KUKA KRL program: dai_sen_calibrate_01.src, dai_sen_calibrate_01.dat

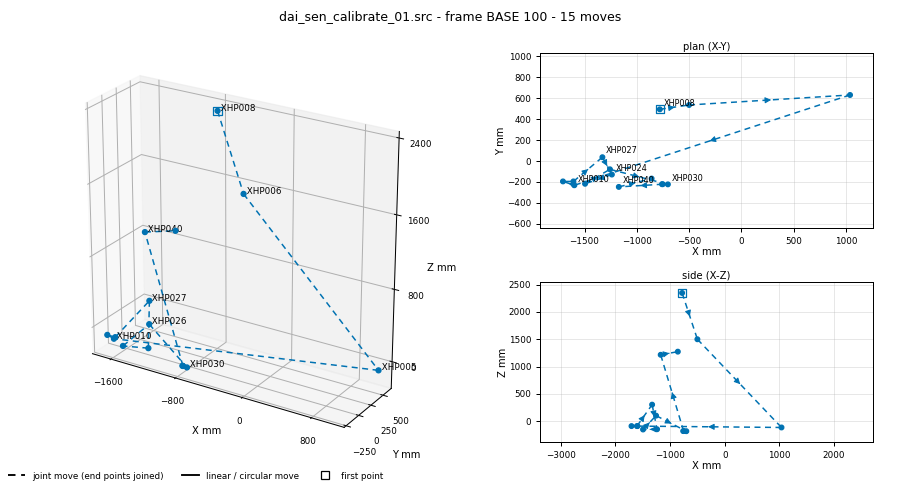
[picture p0: tool path of dai_sen_calibrate_01.src in frame BASE 100, 15 of 17 moves have a stored position in this frame; points joined in program order, loops and branches not executed]
--- dai_sen_calibrate_01.src ---
&ACCESS RVP
&REL 74
&COMMENT Sensopart Kalibrierung
&PARAM TEMPLATE = C:\KRC\roboter\template\vg_appl
&PARAM DISKPATH = KRC:\R1\H_Prog
DEF dai_sen_calibrate_01( )
;FOLD INI;%{PE}
  ;FOLD BASISTECH INI
    GLOBAL INTERRUPT DECL 3 WHEN $STOPMESS==TRUE DO IR_STOPM ( )
    INTERRUPT ON 3
    BAS (#INITMOV,0 )
  ;ENDFOLD (BASISTECH INI)
  ;FOLD USER INI
    ;Make your modifications here
  ;ENDFOLD (USER INI)
;ENDFOLD (INI)
;FOLD ; Anlagenbezeichn: HC51_C    Stations-Nr: 080RB_100;%{PE}
;FOLD Parameters ;%{h}
;Params IlfProvider=kukaroboter.basistech.inlineforms.comments.comment; Kuka.Content=Anlagenbezeichn: HC51_C    Stations-Nr: 080RB_100
;ENDFOLD
;ENDFOLD
;FOLD ; Stand / Version: V1.0;%{PE}
;FOLD Parameters ;%{h}
;Params IlfProvider=kukaroboter.basistech.inlineforms.comments.comment; Kuka.Content=Stand / Version: V1.0
;ENDFOLD
;ENDFOLD
;FOLD ; Name Bearbeiter: EBZ-AE;%{PE}
;FOLD Parameters ;%{h}
;Params IlfProvider=kukaroboter.basistech.inlineforms.comments.comment; Kuka.Content=Name Bearbeiter: EBZ-AE
;ENDFOLD
;ENDFOLD
;FOLD ; Translator Version:29.01.2024 - Version 15.08;%{PE}
;FOLD Parameters ;%{h}
;Params IlfProvider=kukaroboter.basistech.inlineforms.comments.comment; Kuka.Content=Translator Version:29.01.2024 - Version 15.08
;ENDFOLD
;ENDFOLD

;check program once again after mounting calibration plate
WAIT FOR FALSE ;STATUS
;PROGRAM CHECKED BY: SZALA

REPEAT

;FOLD MSG_T1
MSG_SHOW("DAI_H_Prog",#quit,999,"dai_rob_ok_0")
;ENDFOLD

; ***************************************
; A C H T U N G !!! Nur in $T1 abfahren
; ***************************************
UNTIL $T1 == TRUE

REPEAT

;FOLD MSG_T1
MSG_SHOW("DAI_H_Prog",#quit,999,"dai_rob_ok_0")
;ENDFOLD

; ***************************************
; A C H T U N G !!! Nur in $T1 abfahren
; ***************************************
UNTIL $T1 == TRUE

;FOLD PTP HOME Vel=100 % DEFAULT;%{PE}
;FOLD Parameters ;%{h}
;Params IlfProvider=kukaroboter.basistech.inlineforms.movement.old; Kuka.IsGlobalPoint=False; Kuka.PointName=HOME; Kuka.BlendingEnabled=False; Kuka.MoveDataPtpName=DEFAULT; Kuka.VelocityPtp=100; Kuka.CurrentCDSetIndex=0; Kuka.MovementParameterFieldEnabled=True; IlfCommand=PTP
;ENDFOLD
$BWDSTART = FALSE
PDAT_ACT = PDEFAULT
FDAT_ACT = FHOME
BAS(#PTP_PARAMS, 100.0)
SET_CD_PARAMS (0)
PTP XHOME
;ENDFOLD

;Dynamische Pruefung Teil vorhanden
;FOLD PartPresent.CheckOff #1:5279, #2:5280, #3:1025, #4:1025, #5:1025, #6:1025, Bounce Time:100, Constant: Yes;%{PE}%
CheckPartPresent(5279,5280,1025,1025,1025,1025,100, True,FALSE)
;ENDFOLD

;Greifer-Ventile betatigen/pruefen
;FOLD DAI_GripValveCheck.Valve2 State:Fixierstift Ausfahren Gs, 080GRH101-QM1;%{PE}%
CheckValveState(2,1)
;ENDFOLD
;FOLD DAI_GripValveCheck.Valve3 State:Spanner Oeffnen Gs, 080GRH101-QM2;%{PE}%
CheckValveState(3,1)
;ENDFOLD
;FOLD DAI_GripValveCheck.Valve4 State:Sauger Abblasen Gs, 080GRH101-QM3;%{PE}%
CheckValveState(4,1)
;ENDFOLD
;FOLD DAI_GripValveCheck.Valve5 State:Sauger Abblasen Gs, 080GRH101-QM4;%{PE}%
CheckValveState(5,1)
;ENDFOLD

;FOLD PTP HP008 CONT Vel=100 % PDAT16 Tool[110]:MSK_01_XYa_Sensopart Base[100]:SENSOPART_CALIBRATEPLATE ;%{PE}
;FOLD Parameters ;%{h}
;Params IlfProvider=kukaroboter.basistech.inlineforms.movement.old; Kuka.IsGlobalPoint=False; Kuka.PointName=HP008; Kuka.BlendingEnabled=True; Kuka.MoveDataPtpName=PDAT16; Kuka.VelocityPtp=100; Kuka.CurrentCDSetIndex=0; Kuka.MovementParameterFieldEnabled=True; IlfCommand=PTP
;ENDFOLD
$BWDSTART = FALSE
PDAT_ACT = PPDAT16
FDAT_ACT = FHP008
BAS(#PTP_PARAMS, 100.0)
SET_CD_PARAMS (0)
PTP XHP008 C_Dis
;ENDFOLD
;FOLD PTP HP006 CONT Vel=100 % PDAT4 Tool[110]:MSK_01_XYa_Sensopart Base[100]:SENSOPART_CALIBRATEPLATE ;%{PE}
;FOLD Parameters ;%{h}
;Params IlfProvider=kukaroboter.basistech.inlineforms.movement.old; Kuka.IsGlobalPoint=False; Kuka.PointName=HP006; Kuka.BlendingEnabled=True; Kuka.MoveDataPtpName=PDAT4; Kuka.VelocityPtp=100; Kuka.CurrentCDSetIndex=0; Kuka.MovementParameterFieldEnabled=True; IlfCommand=PTP
;ENDFOLD
$BWDSTART = FALSE
PDAT_ACT = PPDAT4
FDAT_ACT = FHP006
BAS(#PTP_PARAMS, 100.0)
SET_CD_PARAMS (0)
PTP XHP006 C_Dis
;ENDFOLD
;FOLD PTP HP005 CONT Vel=100 % PDAT2 Tool[110]:MSK_01_XYa_Sensopart Base[100]:SENSOPART_CALIBRATEPLATE ;%{PE}
;FOLD Parameters ;%{h}
;Params IlfProvider=kukaroboter.basistech.inlineforms.movement.old; Kuka.IsGlobalPoint=False; Kuka.PointName=HP005; Kuka.BlendingEnabled=True; Kuka.MoveDataPtpName=PDAT2; Kuka.VelocityPtp=100; Kuka.CurrentCDSetIndex=0; Kuka.MovementParameterFieldEnabled=True; IlfCommand=PTP
;ENDFOLD
$BWDSTART = FALSE
PDAT_ACT = PPDAT2
FDAT_ACT = FHP005
BAS(#PTP_PARAMS, 100.0)
SET_CD_PARAMS (0)
PTP XHP005 C_Dis
;ENDFOLD

;FOLD PTP HP010 Vel=100 % PDAT3 Tool[110]:MSK_01_XYa_Sensopart Base[100]:SENSOPART_CALIBRATEPLATE ;%{PE}
;FOLD Parameters ;%{h}
;Params IlfProvider=kukaroboter.basistech.inlineforms.movement.old; Kuka.IsGlobalPoint=False; Kuka.PointName=HP010; Kuka.BlendingEnabled=False; Kuka.MoveDataPtpName=PDAT3; Kuka.VelocityPtp=100; Kuka.CurrentCDSetIndex=0; Kuka.MovementParameterFieldEnabled=True; IlfCommand=PTP
;ENDFOLD
$BWDSTART = FALSE
PDAT_ACT = PPDAT3
FDAT_ACT = FHP010
BAS(#PTP_PARAMS, 100.0)
SET_CD_PARAMS (0)
PTP XHP010
;ENDFOLD

;Kalibrationposition
;Fokus-Abstand Kamera zur Kalibrierplatte xx0mm
;FOLD LIN SEN520W080_005 Vel=0.2 m/s CPDAT4 Tool[110]:MSK_01_XYa_Sensopart Base[100]:SENSOPART_CALIBRATEPLATE ;%{PE}
;FOLD Parameters ;%{h}
;Params IlfProvider=kukaroboter.basistech.inlineforms.movement.old; Kuka.IsGlobalPoint=False; Kuka.PointName=SEN520W080_005; Kuka.BlendingEnabled=False; Kuka.MoveDataName=CPDAT4; Kuka.VelocityPath=0.2; Kuka.CurrentCDSetIndex=0; Kuka.MovementParameterFieldEnabled=True; IlfCommand=LIN
;ENDFOLD
$BWDSTART = FALSE
LDAT_ACT = LCPDAT4
FDAT_ACT = FSEN520W080_005
BAS(#CP_PARAMS, 0.2)
SET_CD_PARAMS (0)
LIN XSEN520W080_005
;ENDFOLD

;;FOLD DAI_SEN.CHANGEJOB Cam: 1, Job nbr.: 1 ;%{PE}
; SEN_Cam=1
; SEN_JobResponse=1
; DAI_SEN_CMD ( #ChangeJob )
;;ENDFOLD
;;FOLD DAI_SEN.CALIBRATION Cam: 1, Calibration Base/Tool: 30, Waiting Time: 1 s ;%{PE}
; SEN_CalibMode=2
; SEN_JobResponse=1
; SEN_TimeOut=1
; SEN_CalibBase=30
; SEN_Cam=1
; SEN_CopyMode=1
; DAI_SEN_CMD ( #CALIBRATION )
;;ENDFOLD

;FOLD LIN HP015 Vel=0.2 m/s CPDAT5 Tool[110]:MSK_01_XYa_Sensopart Base[100]:SENSOPART_CALIBRATEPLATE ;%{PE}
;FOLD Parameters ;%{h}
;Params IlfProvider=kukaroboter.basistech.inlineforms.movement.old; Kuka.IsGlobalPoint=False; Kuka.PointName=HP015; Kuka.BlendingEnabled=False; Kuka.MoveDataName=CPDAT5; Kuka.VelocityPath=0.2; Kuka.CurrentCDSetIndex=0; Kuka.MovementParameterFieldEnabled=True; IlfCommand=LIN
;ENDFOLD
$BWDSTART = FALSE
LDAT_ACT = LCPDAT5
FDAT_ACT = FHP015
BAS(#CP_PARAMS, 0.2)
SET_CD_PARAMS (0)
LIN XHP015 C_Dis C_Dis
;ENDFOLD

;FOLD PTP HP027 Vel=100 % PDAT17 Tool[110]:MSK_01_XYa_Sensopart Base[100]:SENSOPART_CALIBRATEPLATE ;%{PE}
;FOLD Parameters ;%{h}
;Params IlfProvider=kukaroboter.basistech.inlineforms.movement.old; Kuka.IsGlobalPoint=False; Kuka.PointName=HP027; Kuka.BlendingEnabled=False; Kuka.MoveDataPtpName=PDAT17; Kuka.VelocityPtp=100; Kuka.CurrentCDSetIndex=0; Kuka.MovementParameterFieldEnabled=True; IlfCommand=PTP
;ENDFOLD
$BWDSTART = FALSE
PDAT_ACT = PPDAT17
FDAT_ACT = FHP027
BAS(#PTP_PARAMS, 100.0)
SET_CD_PARAMS (0)
PTP XHP027
;ENDFOLD
;FOLD PTP HP024 CONT Vel=100 % PDAT14 Tool[110]:MSK_01_XYa_Sensopart Base[100]:SENSOPART_CALIBRATEPLATE ;%{PE}
;FOLD Parameters ;%{h}
;Params IlfProvider=kukaroboter.basistech.inlineforms.movement.old; Kuka.IsGlobalPoint=False; Kuka.PointName=HP024; Kuka.BlendingEnabled=True; Kuka.MoveDataPtpName=PDAT14; Kuka.VelocityPtp=100; Kuka.CurrentCDSetIndex=0; Kuka.MovementParameterFieldEnabled=True; IlfCommand=PTP
;ENDFOLD
$BWDSTART = FALSE
PDAT_ACT = PPDAT14
FDAT_ACT = FHP024
BAS(#PTP_PARAMS, 100.0)
SET_CD_PARAMS (0)
PTP XHP024 C_Dis
;ENDFOLD
;FOLD PTP HP021 CONT Vel=100 % PDAT9 Tool[110]:MSK_01_XYa_Sensopart Base[100]:SENSOPART_CALIBRATEPLATE ;%{PE}
;FOLD Parameters ;%{h}
;Params IlfProvider=kukaroboter.basistech.inlineforms.movement.old; Kuka.IsGlobalPoint=False; Kuka.PointName=HP021; Kuka.BlendingEnabled=True; Kuka.MoveDataPtpName=PDAT9; Kuka.VelocityPtp=100; Kuka.CurrentCDSetIndex=0; Kuka.MovementParameterFieldEnabled=True; IlfCommand=PTP
;ENDFOLD
$BWDSTART = FALSE
PDAT_ACT = PPDAT9
FDAT_ACT = FHP021
BAS(#PTP_PARAMS, 100.0)
SET_CD_PARAMS (0)
PTP XHP021 C_Dis
;ENDFOLD
;FOLD PTP HP026 CONT Vel=100 % PDAT15 Tool[110]:MSK_01_XYa_Sensopart Base[100]:SENSOPART_CALIBRATEPLATE ;%{PE}
;FOLD Parameters ;%{h}
;Params IlfProvider=kukaroboter.basistech.inlineforms.movement.old; Kuka.IsGlobalPoint=False; Kuka.PointName=HP026; Kuka.BlendingEnabled=True; Kuka.MoveDataPtpName=PDAT15; Kuka.VelocityPtp=100; Kuka.CurrentCDSetIndex=0; Kuka.MovementParameterFieldEnabled=True; IlfCommand=PTP
;ENDFOLD
$BWDSTART = FALSE
PDAT_ACT = PPDAT15
FDAT_ACT = FHP026
BAS(#PTP_PARAMS, 100.0)
SET_CD_PARAMS (0)
PTP XHP026 C_Dis
;ENDFOLD
;;FOLD PTP HP020 Vel=100 % PDAT6 Tool[110]:MSK_01_XYa_Sensopart Base[100]:SENSOPART_CALIBRATEPLATE;%{PE}
;;FOLD Parameters ;%{h}
;;Params IlfProvider=kukaroboter.basistech.inlineforms.movement.old; Kuka.IsGlobalPoint=False; Kuka.PointName=HP020; Kuka.BlendingEnabled=False; Kuka.MoveDataPtpName=PDAT6; Kuka.VelocityPtp=100; Kuka.CurrentCDSetIndex=0; Kuka.MovementParameterFieldEnabled=True; IlfCommand=PTP
;;ENDFOLD
;$BWDSTART = FALSE
;PDAT_ACT = PPDAT6
;FDAT_ACT = FHP020
;BAS(#PTP_PARAMS, 100.0)
;SET_CD_PARAMS (0)
;PTP XHP020
;;ENDFOLD
;;FOLD PTP HP025 Vel=100 % PDAT7 Tool[111]:MSK_02_XYa_Sensopart Base[100]:SENSOPART_CALIBRATEPLATE;%{PE}
;;FOLD Parameters ;%{h}
;;Params IlfProvider=kukaroboter.basistech.inlineforms.movement.old; Kuka.IsGlobalPoint=False; Kuka.PointName=HP025; Kuka.BlendingEnabled=False; Kuka.MoveDataPtpName=PDAT7; Kuka.VelocityPtp=100; Kuka.CurrentCDSetIndex=0; Kuka.MovementParameterFieldEnabled=True; IlfCommand=PTP
;;ENDFOLD
;$BWDSTART = FALSE
;PDAT_ACT = PPDAT7
;FDAT_ACT = FHP025
;BAS(#PTP_PARAMS, 100.0)
;SET_CD_PARAMS (0)
;PTP XHP025
;;ENDFOLD
;FOLD PTP HP030 Vel=100 % PDAT8 Tool[111]:MSK_02_XYa_Sensopart Base[100]:SENSOPART_CALIBRATEPLATE;%{PE}
;FOLD Parameters ;%{h}
;Params IlfProvider=kukaroboter.basistech.inlineforms.movement.old; Kuka.IsGlobalPoint=False; Kuka.PointName=HP030; Kuka.BlendingEnabled=False; Kuka.MoveDataPtpName=PDAT8; Kuka.VelocityPtp=100; Kuka.CurrentCDSetIndex=0; Kuka.MovementParameterFieldEnabled=True; IlfCommand=PTP
;ENDFOLD
$BWDSTART = FALSE
PDAT_ACT = PPDAT8
FDAT_ACT = FHP030
BAS(#PTP_PARAMS, 100.0)
SET_CD_PARAMS (0)
PTP XHP030
;ENDFOLD

;Kalibrationposition
;Fokus-Abstand Kamera zur Kalibrierplatte xx0mm
;FOLD LIN SEN520W080_010 Vel=0.2 m/s CPDAT9 Tool[111]:MSK_02_XYa_Sensopart Base[100]:SENSOPART_CALIBRATEPLATE ;%{PE}
;FOLD Parameters ;%{h}
;Params IlfProvider=kukaroboter.basistech.inlineforms.movement.old; Kuka.IsGlobalPoint=False; Kuka.PointName=SEN520W080_010; Kuka.BlendingEnabled=False; Kuka.MoveDataName=CPDAT9; Kuka.VelocityPath=0.2; Kuka.CurrentCDSetIndex=0; Kuka.MovementParameterFieldEnabled=True; IlfCommand=LIN
;ENDFOLD
$BWDSTART = FALSE
LDAT_ACT = LCPDAT9
FDAT_ACT = FSEN520W080_010
BAS(#CP_PARAMS, 0.2)
SET_CD_PARAMS (0)
LIN XSEN520W080_010
;ENDFOLD

;;FOLD DAI_SEN.CHANGEJOB Cam: 1, Job nbr.: 1 ;%{PE}
; SEN_Cam=1
; SEN_JobResponse=1
; DAI_SEN_CMD ( #ChangeJob )
;;ENDFOLD
;;FOLD DAI_SEN.CALIBRATION Cam: 1, Calibration Base/Tool: 30, Waiting Time: 1 s ;%{PE}
; SEN_CalibMode=2
; SEN_JobResponse=1
; SEN_TimeOut=1
; SEN_CalibBase=30
; SEN_Cam=1
; SEN_CopyMode=1
; DAI_SEN_CMD ( #CALIBRATION )
;;ENDFOLD

;FOLD LIN HP035 Vel=0.2 m/s CPDAT10 Tool[111]:MSK_02_XYa_Sensopart Base[100]:SENSOPART_CALIBRATEPLATE ;%{PE}
;FOLD Parameters ;%{h}
;Params IlfProvider=kukaroboter.basistech.inlineforms.movement.old; Kuka.IsGlobalPoint=False; Kuka.PointName=HP035; Kuka.BlendingEnabled=False; Kuka.MoveDataName=CPDAT10; Kuka.VelocityPath=0.2; Kuka.CurrentCDSetIndex=0; Kuka.MovementParameterFieldEnabled=True; IlfCommand=LIN
;ENDFOLD
$BWDSTART = FALSE
LDAT_ACT = LCPDAT10
FDAT_ACT = FHP035
BAS(#CP_PARAMS, 0.2)
SET_CD_PARAMS (0)
LIN XHP035 C_Dis C_Dis
;ENDFOLD

;FOLD PTP HP040 CONT Vel=100 % PDAT11 Tool[111]:MSK_02_XYa_Sensopart Base[100]:SENSOPART_CALIBRATEPLATE ;%{PE}
;FOLD Parameters ;%{h}
;Params IlfProvider=kukaroboter.basistech.inlineforms.movement.old; Kuka.IsGlobalPoint=False; Kuka.PointName=HP040; Kuka.BlendingEnabled=True; Kuka.MoveDataPtpName=PDAT11; Kuka.VelocityPtp=100; Kuka.CurrentCDSetIndex=0; Kuka.MovementParameterFieldEnabled=True; IlfCommand=PTP
;ENDFOLD
$BWDSTART = FALSE
PDAT_ACT = PPDAT11
FDAT_ACT = FHP040
BAS(#PTP_PARAMS, 100.0)
SET_CD_PARAMS (0)
PTP XHP040 C_Dis
;ENDFOLD

;FOLD PTP HP041 CONT Vel=100 % PDAT18 Tool[111]:MSK_02_XYa_Sensopart Base[100]:SENSOPART_CALIBRATEPLATE ;%{PE}
;FOLD Parameters ;%{h}
;Params IlfProvider=kukaroboter.basistech.inlineforms.movement.old; Kuka.IsGlobalPoint=False; Kuka.PointName=HP041; Kuka.BlendingEnabled=True; Kuka.MoveDataPtpName=PDAT18; Kuka.VelocityPtp=100; Kuka.CurrentCDSetIndex=0; Kuka.MovementParameterFieldEnabled=True; IlfCommand=PTP
;ENDFOLD
$BWDSTART = FALSE
PDAT_ACT = PPDAT18
FDAT_ACT = FHP041
BAS(#PTP_PARAMS, 100.0)
SET_CD_PARAMS (0)
PTP XHP041 C_Dis
;ENDFOLD
;FOLD PTP HOME Vel=100 % DEFAULT;%{PE}
;FOLD Parameters ;%{h}
;Params IlfProvider=kukaroboter.basistech.inlineforms.movement.old; Kuka.IsGlobalPoint=False; Kuka.PointName=HOME; Kuka.BlendingEnabled=False; Kuka.MoveDataPtpName=DEFAULT; Kuka.VelocityPtp=100; Kuka.CurrentCDSetIndex=0; Kuka.MovementParameterFieldEnabled=True; IlfCommand=PTP
;ENDFOLD
$BWDSTART = FALSE
PDAT_ACT = PDEFAULT
FDAT_ACT = FHOME
BAS(#PTP_PARAMS, 100.0)
SET_CD_PARAMS (0)
PTP XHOME
;ENDFOLD

;Collision detection - Off
;FOLD COLLDETECT Off ;%{PE}
;FOLD Parameters ;%{h}
;Params IlfProvider=kukaroboter.basistech.inlineforms.colldetect.off; CollDetect.Command=Off
;ENDFOLD
USE_CD_PARAMS(0)
;ENDFOLD

END

--- dai_sen_calibrate_01.dat ---
&ACCESS RVO
&REL 75
&COMMENT Sensopart Kalibrierung
&PARAM TEMPLATE = C:\KRC\roboter\template\vg_appl
&PARAM DISKPATH = KRC:\R1\H_Prog
DEFDAT  DAI_SEN_CALIBRATE_01
;FOLD EXTERNAL DECLARATIONS;%{PE}%MKUKATPBASIS,%CEXT,%VCOMMON,%P
;FOLD BASISTECH EXT;%{PE}%MKUKATPBASIS,%CEXT,%VEXT,%P
EXT  BAS (BAS_COMMAND  :IN,REAL  :IN )
DECL INT SUCCESS
;ENDFOLD (BASISTECH EXT)
;FOLD USER EXT;%{E}%MKUKATPUSER,%CEXT,%VEXT,%P
;Make your modifications here
;ENDFOLD (USER EXT)
;FOLD COLLISION
EXT  COLLSTOP (INT  :IN,INT  :IN )
;ENDFOLD  (Collision)
;ENDFOLD (EXTERNAL DECLERATIONS)
DECL INT handle,answer
; BASIS_SUGG_T declarations
DECL BASIS_SUGG_T LAST_BASIS={POINT1[] "P0                      ",POINT2[] "P0                      ",CP_PARAMS[] "CPDAT0                  ",PTP_PARAMS[] "PDAT0                   ",CONT[] "                        ",CP_VEL[] "2.0                     ",PTP_VEL[] "100                     ",SYNC_PARAMS[] "SYNCDAT                 ",SPL_NAME[] "S0                      ",A_PARAMS[] "ADAT0                   "}
; E6POS declarations
DECL E6POS XHP005={X 1039.35498,Y 631.722290,Z -114.171410,A -93.1388168,B 54.9449844,C -88.7433777,S 18,T 43,E1 -2600.00,E2 0.0,E3 0.0,E4 0.0,E5 0.0,E6 0.0}
DECL E6POS XHP010={X -1596.92566,Y -231.743240,Z -89.1802597,A -89.0549850,B 40.0355186,C -90.0034790,S 18,T 43,E1 -205.766190,E2 0.0,E3 0.0,E4 0.0,E5 0.0,E6 0.0}
DECL E6POS XSEN520W080_005={X -1706.00378,Y -194.999512,Z -89.0078659,A -89.9999695,B 39.9999504,C -90.0001526,S 18,T 11,E1 -200.000,E2 0.0,E3 0.0,E4 0.0,E5 0.0,E6 0.0}
DECL E6POS XHP015={X -1606.01636,Y -195.001434,Z -89.0170746,A -89.9999695,B 39.9999466,C -90.0001602,S 18,T 11,E1 -200.000,E2 0.0,E3 0.0,E4 0.0,E5 0.0,E6 0.0}
DECL E6POS XHP020={X -613.699,Y 127.543434,Z 25.9875164,A -160.751953,B 84.9972763,C -160.752335,S 18,T 11,E1 -1727.58594,E2 0.0,E3 0.0,E4 0.0,E5 0.0,E6 0.0}
DECL E6POS XHP025={X -850.755310,Y -176.272644,Z -270.095642,A 94.6133957,B 68.1071396,C 97.6182480,S 18,T 3,E1 -1393.04382,E2 0.0,E3 0.0,E4 0.0,E5 0.0,E6 0.0}
DECL E6POS XHP030={X -702.608032,Y -223.037415,Z -182.485916,A 93.7805176,B 64.4597092,C 95.9692688,S 18,T 3,E1 -1804.39478,E2 0.0,E3 0.0,E4 0.0,E5 0.0,E6 0.0}
DECL E6POS XSEN520W080_010={X -758.821960,Y -221.478745,Z -179.963364,A 93.7783051,B 64.4603958,C 95.9665756,S 18,T 3,E1 -1804.39478,E2 0.0,E3 0.0,E4 0.0,E5 0.0,E6 0.0}
DECL E6POS XHP035={X -751.937561,Y -221.671463,Z -180.272858,A 93.7785950,B 64.4602661,C 95.9668503,S 18,T 3,E1 -1804.39478,E2 0.0,E3 0.0,E4 0.0,E5 0.0,E6 0.0}
DECL E6POS XHP040={X -1171.95508,Y -247.432,Z 1216.19019,A 177.204666,B 36.6067238,C -34.5377922,S 18,T 3,E1 -2533.72266,E2 0.0,E3 0.0,E4 0.0,E5 0.0,E6 0.0}
; FDAT declarations
DECL FDAT FHOME={TOOL_NO 110,BASE_NO 100,IPO_FRAME #BASE,POINT2[] " "}
DECL FDAT FHP005={TOOL_NO 110,BASE_NO 100,IPO_FRAME #BASE,POINT2[] " "}
DECL FDAT FHP010={TOOL_NO 110,BASE_NO 100,IPO_FRAME #BASE,POINT2[] " "}
DECL FDAT FSEN520W080_005={TOOL_NO 110,BASE_NO 100,IPO_FRAME #BASE,POINT2[] " "}
DECL FDAT FHP015={TOOL_NO 110,BASE_NO 100,IPO_FRAME #BASE,POINT2[] " "}
DECL FDAT FHP020={TOOL_NO 110,BASE_NO 100,IPO_FRAME #BASE,POINT2[] " "}
DECL FDAT FHP025={TOOL_NO 111,BASE_NO 100,IPO_FRAME #BASE,POINT2[] " "}
DECL FDAT FHP030={TOOL_NO 111,BASE_NO 100,IPO_FRAME #BASE,POINT2[] " "}
DECL FDAT FSEN520W080_010={TOOL_NO 111,BASE_NO 100,IPO_FRAME #BASE,POINT2[] " "}
DECL FDAT FHP035={TOOL_NO 111,BASE_NO 100,IPO_FRAME #BASE,POINT2[] " "}
DECL FDAT FHP040={TOOL_NO 111,BASE_NO 100,IPO_FRAME #BASE,POINT2[] " "}
; LDAT declarations
DECL LDAT LCPDAT4={VEL 0.200000,ACC 100.000,APO_DIST 0.0,APO_FAC 50.0000,AXIS_VEL 100.000,AXIS_ACC 100.000,ORI_TYP #VAR,CIRC_TYP #BASE,JERK_FAC 50.0000,GEAR_JERK 50.0000,EXAX_IGN 0}
DECL LDAT LCPDAT5={VEL 0.200000,ACC 100.000,APO_DIST 0.0,APO_FAC 50.0000,AXIS_VEL 100.000,AXIS_ACC 100.000,ORI_TYP #VAR,CIRC_TYP #BASE,JERK_FAC 50.0000,GEAR_JERK 50.0000,EXAX_IGN 0}
DECL LDAT LCPDAT9={VEL 0.200000,ACC 100.000,APO_DIST 0.0,APO_FAC 50.0000,AXIS_VEL 100.000,AXIS_ACC 100.000,ORI_TYP #VAR,CIRC_TYP #BASE,JERK_FAC 50.0000,GEAR_JERK 50.0000,EXAX_IGN 0}
DECL LDAT LCPDAT10={VEL 0.200000,ACC 100.000,APO_DIST 0.0,APO_FAC 50.0000,AXIS_VEL 100.000,AXIS_ACC 100.000,ORI_TYP #VAR,CIRC_TYP #BASE,JERK_FAC 50.0000,GEAR_JERK 50.0000,EXAX_IGN 0}
; PDAT declarations
DECL PDAT PPDAT2={VEL 100.000,ACC 100.000,APO_DIST 0.0,APO_MODE #CDIS,GEAR_JERK 50.0000,EXAX_IGN 0}
DECL PDAT PPDAT6={VEL 100.000,ACC 100.000,APO_DIST 0.0,APO_MODE #CDIS,GEAR_JERK 50.0000,EXAX_IGN 0}
DECL PDAT PPDAT7={VEL 100.000,ACC 100.000,APO_DIST 0.0,APO_MODE #CDIS,GEAR_JERK 50.0000,EXAX_IGN 0}
DECL PDAT PPDAT8={VEL 100.000,ACC 100.000,APO_DIST 0.0,APO_MODE #CDIS,GEAR_JERK 50.0000,EXAX_IGN 0}
DECL PDAT PPDAT11={VEL 100.000,ACC 100.000,APO_DIST 0.0,APO_MODE #CDIS,GEAR_JERK 50.0000,EXAX_IGN 0}

DECL MODULEPARAM_T LAST_TP_PARAMS={PARAMS[] "Kuka.PointName=HP026; Kuka.FrameData.base_no=100; Kuka.FrameData.tool_no=110; Kuka.FrameData.ipo_frame=#BASE; Kuka.FrameData.point2=; Kuka.isglobalpoint=False; Kuka.MoveDataName=CPDAT3; Kuka.MovementData.cb={AUX_PT {ORI #CONSIDER,E1 #CONSIDER,E2 #CONSIDER,E3 #CONSIDER,E4 #CONSIDER,E5 #CONSIDER,E6 #CONSIDER},TARGET_PT {ORI #INTERPOLATE,E1 #INTERPOLATE,E2 #INTERPOLATE,E3 #INTERPOLATE,E4 #INTERPOLATE,E5 #INTERPOLATE,E6 #INTERPOLATE}}; Kuka.MovementData.apo_fac=50; Kuka.MovementData.apo_dist=0; Kuka.MovementData.axis_acc=100; Kuka.MovementData.axis_vel=100; Kuka.MovementData.circ_typ=#BASE; Kuka.MovementData.jerk_fac=50; Kuka.MovementData.ori_typ=#VAR; Kuka.MovementData.vel=100; Kuka.MovementData.acc=100; Kuka.MovementData.exax_ign=0; Kuka.VelocityPath=0.2; Kuka.BlendingEnabled=True; Kuka.APXEnabled=False; Kuka.CurrentCDSetIndex=0; Kuka.MoveDataPtpName=PDAT15; Kuka.MovementDataPdat.apo_mode=#CDIS; Kuka.MovementDataPdat.apo_dist=0; Kuka.VelocityPtp=100  "}
DECL PDAT PPDAT3={VEL 100.000,ACC 100.000,APO_DIST 500.000,APO_MODE #CDIS,GEAR_JERK 100.000,EXAX_IGN 0}
DECL E6POS XHP006={X -500.103027,Y 536.082031,Z 1500.19922,A -169.213425,B 34.4071426,C 149.267273,S 18,T 43,E1 -2600.00,E2 0.0,E3 0.0,E4 0.0,E5 0.0,E6 0.0}
DECL FDAT FHP006={TOOL_NO 110,BASE_NO 100,IPO_FRAME #BASE,POINT2[] " "}
DECL PDAT PPDAT4={VEL 100.000,ACC 100.000,APO_DIST 0.0,APO_MODE #CDIS,GEAR_JERK 50.0000,EXAX_IGN 0}
DECL E6POS XHP021={X -1494.82141,Y -217.606430,Z -151.342239,A -93.8292694,B 73.7935410,C 125.149315,S 18,T 43,E1 -1655.5,E2 0.0,E3 0.0,E4 0.0,E5 0.0,E6 0.0}
DECL FDAT FHP021={TOOL_NO 110,BASE_NO 100,IPO_FRAME #BASE,POINT2[] " "}
DECL PDAT PPDAT9={VEL 100.000,ACC 100.000,APO_DIST 0.0,APO_MODE #CDIS,GEAR_JERK 50.0000,EXAX_IGN 0}
DECL E6POS XHP024={X -1238.38416,Y -129.298340,Z -146.615417,A -106.528198,B 71.9078445,C 131.198242,S 18,T 43,E1 -1655.5,E2 0.0,E3 0.0,E4 0.0,E5 0.0,E6 0.0}
DECL FDAT FHP024={TOOL_NO 110,BASE_NO 100,IPO_FRAME #BASE,POINT2[] " "}
DECL PDAT PPDAT14={VEL 100.000,ACC 100.000,APO_DIST 0.0,APO_MODE #CDIS,GEAR_JERK 50.0000,EXAX_IGN 0}
DECL E6POS XHP026={X -1256.61169,Y -79.1451721,Z 102.527336,A -163.508835,B 67.4663391,C 23.6411324,S 18,T 11,E1 -1655.5,E2 0.0,E3 0.0,E4 0.0,E5 0.0,E6 0.0}
DECL FDAT FHP026={TOOL_NO 110,BASE_NO 100,IPO_FRAME #BASE,POINT2[] " "}
DECL PDAT PPDAT15={VEL 100.000,ACC 100.000,APO_DIST 0.0,APO_MODE #CDIS,GEAR_JERK 50.0000,EXAX_IGN 0}
DECL E6POS XHP008={X -779.686707,Y 494.498138,Z 2348.19873,A -175.757126,B 17.4712486,C 131.541367,S 18,T 43,E1 -2600.00,E2 0.0,E3 0.0,E4 0.0,E5 0.0,E6 0.0}
DECL FDAT FHP008={TOOL_NO 110,BASE_NO 100,IPO_FRAME #BASE,POINT2[] " "}
DECL PDAT PPDAT16={VEL 100.000,ACC 100.000,APO_DIST 0.0,APO_MODE #CDIS,GEAR_JERK 50.0000,EXAX_IGN 0}
DECL E6POS XHP027={X -1328.82031,Y 36.4979591,Z 303.547607,A -152.226929,B 60.2146683,C 96.8618393,S 18,T 43,E1 -1655.49500,E2 0.0,E3 0.0,E4 0.0,E5 0.0,E6 0.0}
DECL FDAT FHP027={TOOL_NO 110,BASE_NO 100,IPO_FRAME #BASE,POINT2[] " "}
DECL PDAT PPDAT17={VEL 100.000,ACC 100.000,APO_DIST 0.0,APO_MODE #CDIS,GEAR_JERK 50.0000,EXAX_IGN 0}
DECL E6POS XHP041={X -858.235596,Y -167.701965,Z 1273.29370,A 176.900055,B 34.6555328,C -12.6553259,S 18,T 35,E1 -2620.65845,E2 0.0,E3 0.0,E4 0.0,E5 0.0,E6 0.0}
DECL FDAT FHP041={TOOL_NO 111,BASE_NO 100,IPO_FRAME #BASE,POINT2[] " "}
DECL PDAT PPDAT18={VEL 100.000,ACC 100.000,APO_DIST 0.0,APO_MODE #CDIS,GEAR_JERK 50.0000,EXAX_IGN 0}
ENDDAT
